// TIA Portal V17 export
// export: Created 2021-12-03T08:13:04.2830787Z, ExportSetting WithDefaults, DisplayName Totally Integrated Automation Portal, DisplayVersion V17, DisplayName TIA Portal Openness, DisplayVersion V17, DisplayName TIA Portal Version Control Interface, DisplayVersion V17, DisplayName STEP 7 Professional, DisplayVersion V17, DisplayName STEP 7 Safety, DisplayVersion V17, DisplayName WinCC Advanced, DisplayVersion V17
FUNCTION "FC_ConvCtrl" : Void   // FC500, FBD
VERSION : 0.1
// stored: AutoNumber false, IsIECCheckEnabled false, UDAEnableTagReadback false
   VAR_TEMP
      TimeMowBack : Int;
      SRStartCountTime : Bool;
      PSConvStpBwd : Bool;
      PSConvXRayBwd : Bool;
      P_SpeedSave : Bool;
      TimeMowFwdReal : Word;
      PSConvStpFwd : Bool;
      NPSConvStpFwd : Bool;
      NPSConvXRayFwd : Bool;
      End : Bool;
      PPSConvStpBwd : Bool;
   END_VAR
   VAR CONSTANT
      TimeMowFwd : Int := 1;
   END_VAR
   VAR_TEMP   // added for the SCL form of the ladder/FBD networks
      _w1 : Bool;
   END_VAR
BEGIN

REGION Network 1: Включение частотного преобразователя
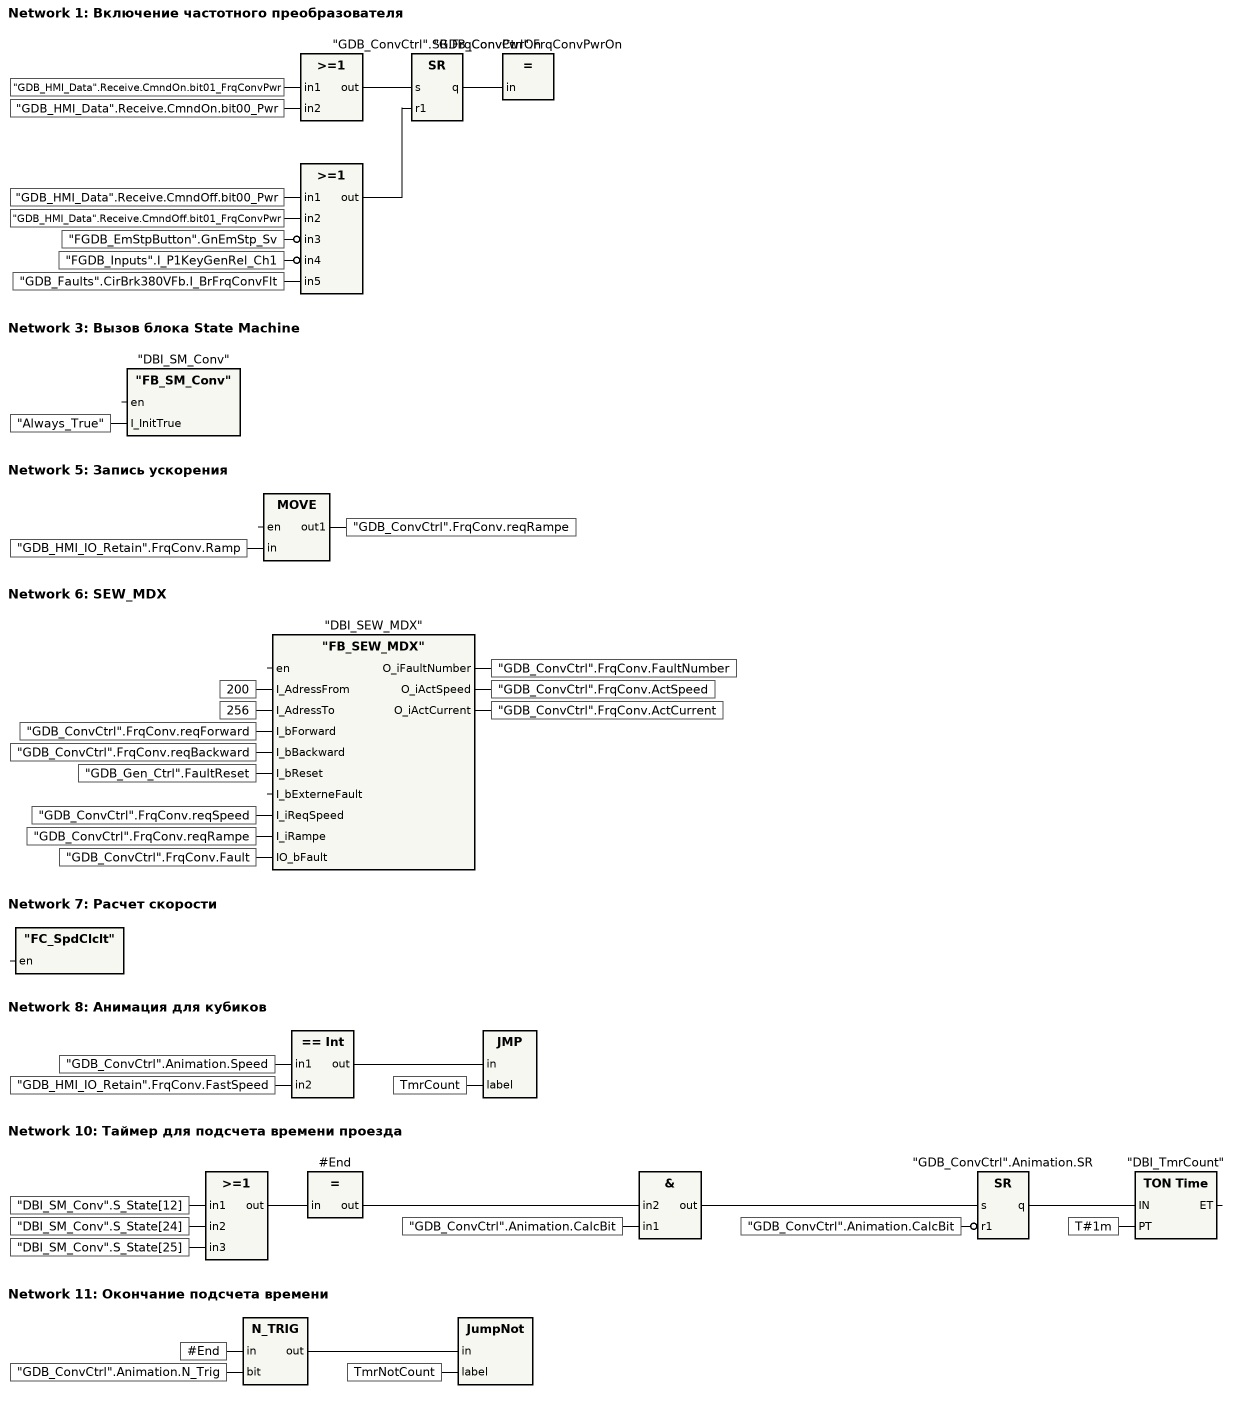
   IF "GDB_HMI_Data".Receive.CmndOn.bit01_FrqConvPwr OR "GDB_HMI_Data".Receive.CmndOn.bit00_Pwr THEN
       "GDB_ConvCtrl".SR.FrqConvPwrOn := TRUE;   // SR flip-flop
   END_IF;
   IF "GDB_HMI_Data".Receive.CmndOff.bit00_Pwr OR "GDB_HMI_Data".Receive.CmndOff.bit01_FrqConvPwr OR NOT "FGDB_EmStpButton".GnEmStp_Sv OR NOT "FGDB_Inputs".I_P1KeyGenRel_Ch1 OR "GDB_Faults".CirBrk380VFb.I_BrFrqConvFlt THEN
       "GDB_ConvCtrl".SR.FrqConvPwrOn := FALSE;
   END_IF;
   "GDB_ConvCtrl".FrqConvPwrOn := "GDB_ConvCtrl".SR.FrqConvPwrOn;
END_REGION

NETWORK
TITLE = Условия перехода для конвейера
// Fct.-Name : TRUE
      A     "GDB_Gen_Ctrl".Restart;
      =     "DBI_SM_Conv".S_Conditions[1];

// Fct.-Name : Frq Conv Power is On
      AN    "FGDB_Inputs".I_FBPowerConveyor;
      =     "DBI_SM_Conv".S_Conditions[2];

// Fct.-Name : /Frq Conv Power is On
      AN    "DBI_SM_Conv".S_Conditions[2];
      =     "DBI_SM_Conv".S_Conditions[3];

// Fct.-Name : Frq Conv Fault
      A     "GDB_ConvCtrl".FrqConv.Fault;
      AN    "GDB_HMI_Data".Receive.Simulation.Console_SimEn;
      =     "DBI_SM_Conv".S_Conditions[4];

// Fct.-Name : STO Drive
      X     "GDB_Inputs".I_P2ConvLocal;
      X     "FGDB_Safety_Perimeter".SAreaClose;
      =     "DBI_SM_Conv".S_Conditions[5];

// Fct.-Name : STO Drive
      AN    "DBI_SM_Conv".S_Conditions[5];
      =     "DBI_SM_Conv".S_Conditions[6];

// Fct.-Name : Conv is Forward Stop Position
      A     "GDB_Inputs".I_PSConvStpFwd;
      =     "DBI_SM_Conv".S_Conditions[9];

// Fct.-Name : Conv is Backward Stop Position
      A     "GDB_Inputs".I_PSConvStpBwd;
      =     "DBI_SM_Conv".S_Conditions[10];

// Fct.-Name : Auto Conv Forward Move
      O     "GDB_ScanSequence".Action.FwdMoveReq;
      O     "GDB_HmiTestBtns".TB1_08_ConvFwrd;
      O     "GDB_SpdClclt".Action.Homming;
      FP    "GDB_ConvCtrl".Trig.P_StrtFwd;
      =     "DBI_SM_Conv".S_Conditions[11];

// Fct.-Name : Auto Conv Backward Move
      O     "GDB_ScanSequence".Action.BwdMoveReq;
      O     "GDB_HmiTestBtns".TB1_09_ConvBwrd;
      O     "GDB_SpdClclt".Action.BwdStrt;
      FP    "GDB_ConvCtrl".Trig.P_StrtBwd;
      =     "DBI_SM_Conv".S_Conditions[12];

// Fct.-Name : Conv Stop
      O     "GDB_ScanSequence".IntrptCycl;
      O     "GDB_Faults".Conveyer.FrqConv;
      O     "GDB_Faults".Conveyer.CycleTime;
      =     "DBI_SM_Conv".S_Conditions[14];

// Fct.-Name : Ack Fault
      A     "GDB_Gen_Ctrl".FaultReset;
      =     "DBI_SM_Conv".S_Conditions[15];

// Fct.-Name : Conv JogMode selected
      A     "GDB_Inputs".I_P2ConvLocal;
      =     "DBI_SM_Conv".S_Conditions[16];

// Fct.-Name : /Conv JogMode selected
      AN    "DBI_SM_Conv".S_Conditions[16];
      =     "DBI_SM_Conv".S_Conditions[17];

// Fct.-Name : Conv Agree B
      A     "GDB_Inputs".I_P2ConvLocal;
      A     "FGDB_Inputs".I_P2AgreeBut_Ch1;
      =     "DBI_SM_Conv".S_Conditions[18];

// Fct.-Name : /Conv Agree B
      AN    "DBI_SM_Conv".S_Conditions[18];
      =     "DBI_SM_Conv".S_Conditions[19];

// Fct.-Name : Conv Jog Fwd
      A     "GDB_Inputs".I_P2ConvLocal;
      A     "GDB_Inputs".I_P2ConvFwd;
      =     "DBI_SM_Conv".S_Conditions[20];

// Fct.-Name : /Conv Jog Fwd
      AN    "DBI_SM_Conv".S_Conditions[20];
      =     "DBI_SM_Conv".S_Conditions[21];

// Fct.-Name : Conv Jog Bwd
      A     "GDB_Inputs".I_P2ConvLocal;
      A     "GDB_Inputs".I_P2ConvBwd;
      =     "DBI_SM_Conv".S_Conditions[22];

// Fct.-Name : /Conv Jog Bwd
      AN    "DBI_SM_Conv".S_Conditions[22];
      =     "DBI_SM_Conv".S_Conditions[23];

// Fct.-Name : Conv Fast Forward
      A     "GDB_Inputs".I_PSConvSlowBwd;
      FN    "GDB_ConvCtrl".Trig.N_SlowBwd;
      =     "DBI_SM_Conv".S_Conditions[25];

// Fct.-Name : Conv Slow Forward
      A     "GDB_Inputs".I_PSConvSlowFwd;
      FP    "GDB_ConvCtrl".Trig.P_SlowFwd;
      =     "DBI_SM_Conv".S_Conditions[26];

// Fct.-Name : Conv Fast Backward
      A     "GDB_Inputs".I_PSConvSlowFwd;
      FN    "GDB_ConvCtrl".Trig.N_SlowFwd;
      =     "DBI_SM_Conv".S_Conditions[27];

// Fct.-Name : Conv Slow Backward
      A     "GDB_Inputs".I_PSConvSlowBwd;
      FP    "GDB_ConvCtrl".Trig.P_SlowBwd;
      =     "DBI_SM_Conv".S_Conditions[28];



REGION Network 3: Вызов блока State Machine
   "DBI_SM_Conv"(I_InitTrue := "Always_True");   // "FB_SM_Conv"
END_REGION

NETWORK
TITLE = Выбор направления и скорости
// Forward
      O     "DBI_SM_Conv".S_State[10];
      O     "DBI_SM_Conv".S_State[16];
      O     "DBI_SM_Conv".S_State[22];
      O     "DBI_SM_Conv".S_State[23];
      =     "GDB_ConvCtrl".FrqConv.reqForward;

// Backward
      O     "DBI_SM_Conv".S_State[12];
      O     "DBI_SM_Conv".S_State[18];
      O     "DBI_SM_Conv".S_State[24];
      O     "DBI_SM_Conv".S_State[25];
      =     "GDB_ConvCtrl".FrqConv.reqBackward;

// Speed
      O     "DBI_SM_Conv".S_State[10];
      O     "DBI_SM_Conv".S_State[12];
      O     "DBI_SM_Conv".S_State[16];
      O     "DBI_SM_Conv".S_State[18];
      O     "DBI_SM_Conv".S_State[23];
      O     "DBI_SM_Conv".S_State[24];
      JCN   SpdS;
      L     "GDB_HMI_IO_Retain".FrqConv.LowSpeed;
      T     "GDB_ConvCtrl".FrqConv.reqSpeed;
      JU    SpdE;
SpdS: NOP   0;

      O     "DBI_SM_Conv".S_State[22];
      O     "DBI_SM_Conv".S_State[25];
      JCN   SpdF;
      L     "GDB_HMI_IO_Retain".FrqConv.FastSpeed;
      T     "GDB_ConvCtrl".FrqConv.reqSpeed;
      JU    SpdE;
SpdF: NOP   0;
      L     0;
      T     "GDB_ConvCtrl".FrqConv.reqSpeed;
SpdE: NOP   0;

REGION Network 5: Запись ускорения
   "GDB_ConvCtrl".FrqConv.reqRampe := "GDB_HMI_IO_Retain".FrqConv.Ramp;
END_REGION

REGION Network 6: SEW_MDX
   "DBI_SEW_MDX"(I_AdressFrom := 200,   // "FB_SEW_MDX"
                 I_AdressTo := 256,
                 I_bForward := "GDB_ConvCtrl".FrqConv.reqForward,
                 I_bBackward := "GDB_ConvCtrl".FrqConv.reqBackward,
                 I_bReset := "GDB_Gen_Ctrl".FaultReset,
                 I_iReqSpeed := "GDB_ConvCtrl".FrqConv.reqSpeed,
                 I_iRampe := "GDB_ConvCtrl".FrqConv.reqRampe,
                 IO_bFault := "GDB_ConvCtrl".FrqConv.Fault,
                 O_iFaultNumber => "GDB_ConvCtrl".FrqConv.FaultNumber,
                 O_iActSpeed => "GDB_ConvCtrl".FrqConv.ActSpeed,
                 O_iActCurrent => "GDB_ConvCtrl".FrqConv.ActCurrent);
END_REGION

REGION Network 7: Расчет скорости
   "FC_SpdClclt"();
END_REGION

REGION Network 8: Анимация для кубиков
   IF "GDB_ConvCtrl".Animation.Speed = "GDB_HMI_IO_Retain".FrqConv.FastSpeed THEN GOTO TmrCount; END_IF;
END_REGION

NETWORK
TITLE = Взведение бита
      L     "GDB_HMI_IO_Retain".FrqConv.FastSpeed;
      T     "GDB_ConvCtrl".Animation.Speed;

      S     "GDB_ConvCtrl".Animation.CalcBit;

REGION Network 10: Таймер для подсчета времени проезда
   TmrCount:
   #End := "DBI_SM_Conv".S_State[12] OR "DBI_SM_Conv".S_State[24] OR "DBI_SM_Conv".S_State[25];
   IF #End AND "GDB_ConvCtrl".Animation.CalcBit THEN
       "GDB_ConvCtrl".Animation.SR := TRUE;   // SR flip-flop
   END_IF;
   IF NOT "GDB_ConvCtrl".Animation.CalcBit THEN "GDB_ConvCtrl".Animation.SR := FALSE; END_IF;
   "DBI_TmrCount".TON(IN := "GDB_ConvCtrl".Animation.SR, PT := T#1m);
END_REGION

REGION Network 11: Окончание подсчета времени
   // no SCL statement known for JumpNot: written as a call
   #_w1 := NOT #End AND "GDB_ConvCtrl".Animation.N_Trig;   // falling edge
   "GDB_ConvCtrl".Animation.N_Trig := #End;
   JumpNot(in := #_w1, label := TmrNotCount);
END_REGION

NETWORK
TITLE = Сброс бита
      L     "DBI_TmrCount".ET;
      T     "GDB_HMI_IO_Retain".TmrValue;

      R     "GDB_ConvCtrl".Animation.CalcBit;

REGION Network 13: Таймер для анимации
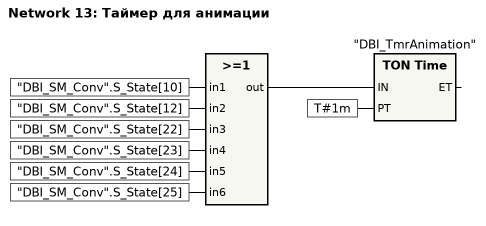
   TmrNotCount:
   "DBI_TmrAnimation".TON(IN := "DBI_SM_Conv".S_State[10] OR "DBI_SM_Conv".S_State[12] OR "DBI_SM_Conv".S_State[22] OR "DBI_SM_Conv".S_State[23] OR "DBI_SM_Conv".S_State[24] OR "DBI_SM_Conv".S_State[25],
                          PT := T#1m);
END_REGION

NETWORK
TITLE = 
      L     "DBI_TmrAnimation".ET;
      L     "GDB_HMI_IO_Retain".TmrValue;
      /R;
      T     "GDB_ConvCtrl".Animation.Value;
END_FUNCTION
